{attribute 'qualified_only'}
VAR_GLOBAL
	fTooltipXCoordGlobalIni: LREAL := 2.8;
	fTooltipYCoordGlobalIni: LREAL := 2.2;
	
	fTheta1 : LREAL := 0;
	fAngleMainArmInverse :	LREAL;
	fAngleKnuckleArmInverse : LREAL;
	fStrokeActuatorMainInverse : LREAL;
	fStrokeActuatorKnuckleInverse : LREAL;
END_VAR

(* stored: Version 1.1.0.1, ProductVersion 3.1.4024.12
   GVL GVL_InverseKinematics: Id {fd34d786-3bd4-452e-849d-6618ad2b1310} *)
